Fanuc KAREL source: KA00224.KL

PROGRAM KA00224
%NOLOCKGROUP
VAR
  SRC: ARRAY[4] OF JOINTPOS
  DST: ARRAY[4] OF XYZWPR
BEGIN
  DST = SRC
END KA00224
